    |   movel([0.097941, -1.446408, -2.526251, -0.739730, 1.570796, 1.668738],accel_mss,speed_ms,0,blend_radius_m)
    |   movel([0.099075, -1.445086, -2.527311, -0.739992, 1.570796, 1.669872],accel_mss,speed_ms,0,blend_radius_m)
    |   movel([0.103315, -1.440776, -2.530747, -0.740866, 1.570796, 1.674111],accel_mss,speed_ms,0,blend_radius_m)
    |   movel([0.107663, -1.436494, -2.534133, -0.741762, 1.570796, 1.678459],accel_mss,speed_ms,0,blend_radius_m)
    |   movel([0.104362, -1.438461, -2.532581, -0.741347, 1.570796, 1.675158],accel_mss,speed_ms,0,blend_radius_m)
    |   movel([0.101406, -1.440513, -2.530956, -0.740920, 1.570796, 1.672202],accel_mss,speed_ms,0,blend_radius_m)
    |   movel([0.098613, -1.442794, -2.529142, -0.740453, 1.570796, 1.669409],accel_mss,speed_ms,0,blend_radius_m)
    |   movel([0.095804, -1.445440, -2.527027, -0.739922, 1.570796, 1.666601],accel_mss,speed_ms,0,blend_radius_m)
    |   movel([0.097126, -1.443984, -2.528192, -0.740213, 1.570796, 1.667922],accel_mss,speed_ms,0,blend_radius_m)
    |   movel([0.098287, -1.442464, -2.529404, -0.740520, 1.570796, 1.669083],accel_mss,speed_ms,0,blend_radius_m)
    |   movel([0.102381, -1.436114, -2.534433, -0.741843, 1.570796, 1.673177],accel_mss,speed_ms,0,blend_radius_m)
    |   movel([0.103529, -1.434547, -2.535663, -0.742178, 1.570796, 1.674326],accel_mss,speed_ms,0,blend_radius_m)
    |   movel([0.104838, -1.433026, -2.536855, -0.742508, 1.570796, 1.675635],accel_mss,speed_ms,0,blend_radius_m)
    |   movel([0.106771, -1.431152, -2.538318, -0.742919, 1.570796, 1.677568],accel_mss,speed_ms,0,blend_radius_m)
    |   movel([0.108499, -1.429865, -2.539320, -0.743204, 1.570796, 1.679295],accel_mss,speed_ms,0,blend_radius_m)
    |   movel([0.108872, -1.429473, -2.539624, -0.743291, 1.570796, 1.679668],accel_mss,speed_ms,0,blend_radius_m)
    |   movel([0.108963, -1.429084, -2.539927, -0.743378, 1.570796, 1.679759],accel_mss,speed_ms,0,blend_radius_m)
    |   movel([0.108687, -1.428925, -2.540050, -0.743414, 1.570796, 1.679484],accel_mss,speed_ms,0,blend_radius_m)
    |   movel([0.108143, -1.428947, -2.540033, -0.743409, 1.570796, 1.678940],accel_mss,speed_ms,0,blend_radius_m)
    |   movel([0.107429, -1.429105, -2.539910, -0.743374, 1.570796, 1.678225],accel_mss,speed_ms,0,blend_radius_m)
    |   movel([0.105873, -1.429619, -2.539511, -0.743259, 1.570796, 1.676669],accel_mss,speed_ms,0,blend_radius_m)
    |   movel([0.104794, -1.430074, -2.539157, -0.743158, 1.570796, 1.675591],accel_mss,speed_ms,0,blend_radius_m)
    |   movel([0.106351, -1.428336, -2.540507, -0.743546, 1.570796, 1.677147],accel_mss,speed_ms,0,blend_radius_m)
    |   movel([0.108214, -1.426670, -2.541796, -0.743923, 1.570796, 1.679010],accel_mss,speed_ms,0,blend_radius_m)
    |   movel([0.112152, -1.423648, -2.544124, -0.744617, 1.570796, 1.682948],accel_mss,speed_ms,0,blend_radius_m)
    |   speed_ms = 0.005
    |   movel([0.112152, -1.415184, -2.540319, -0.756886, 1.570796, 1.682948],accel_mss,speed_ms,0,blend_radius_m)
    |   speed_ms = 0.040
    |   movel([0.104332, -1.417020, -2.538925, -0.756444, 1.570796, 1.675128],accel_mss,speed_ms,0,blend_radius_m)
    |   speed_ms = 0.005
    |   movel([0.104332, -1.425469, -2.542723, -0.744197, 1.570796, 1.675128],accel_mss,speed_ms,0,blend_radius_m)
    |   speed_ms = 0.025
    |   movel([0.103555, -1.424729, -2.543293, -0.744367, 1.570796, 1.674352],accel_mss,speed_ms,0,blend_radius_m)
    |   movel([0.102591, -1.424211, -2.543692, -0.744487, 1.570796, 1.673387],accel_mss,speed_ms,0,blend_radius_m)
    |   movel([0.101472, -1.423893, -2.543936, -0.744560, 1.570796, 1.672268],accel_mss,speed_ms,0,blend_radius_m)
    |   movel([0.100232, -1.423752, -2.544044, -0.744593, 1.570796, 1.671028],accel_mss,speed_ms,0,blend_radius_m)
    |   movel([0.098900, -1.423771, -2.544029, -0.744588, 1.570796, 1.669696],accel_mss,speed_ms,0,blend_radius_m)
    |   movel([0.097513, -1.423927, -2.543910, -0.744552, 1.570796, 1.668309],accel_mss,speed_ms,0,blend_radius_m)
    |   movel([0.094694, -1.424556, -2.543426, -0.744407, 1.570796, 1.665490],accel_mss,speed_ms,0,blend_radius_m)
    |   speed_ms = 0.005
    |   movel([0.094694, -1.416100, -2.539624, -0.756665, 1.570796, 1.665490],accel_mss,speed_ms,0,blend_radius_m)
    |   speed_ms = 0.040
    |   movel([0.105862, -1.410628, -2.543757, -0.758004, 1.570796, 1.676658],accel_mss,speed_ms,0,blend_radius_m)
    |   speed_ms = 0.005
    |   movel([0.105862, -1.419125, -2.547582, -0.745682, 1.570796, 1.676658],accel_mss,speed_ms,0,blend_radius_m)
    |   speed_ms = 0.025
    |   movel([0.105216, -1.417553, -2.548777, -0.746059, 1.570796, 1.676012],accel_mss,speed_ms,0,blend_radius_m)
    |   movel([0.104462, -1.416106, -2.549874, -0.746409, 1.570796, 1.675259],accel_mss,speed_ms,0,blend_radius_m)
    |   movel([0.103559, -1.414829, -2.550839, -0.746721, 1.570796, 1.674355],accel_mss,speed_ms,0,blend_radius_m)
    |   movel([0.102461, -1.413767, -2.551639, -0.746983, 1.570796, 1.673258],accel_mss,speed_ms,0,blend_radius_m)
    |   movel([0.101125, -1.412972, -2.552238, -0.747179, 1.570796, 1.671921],accel_mss,speed_ms,0,blend_radius_m)
    |   movel([0.099510, -1.412483, -2.552605, -0.747301, 1.570796, 1.670307],accel_mss,speed_ms,0,blend_radius_m)
    |   movel([0.097573, -1.412353, -2.552703, -0.747333, 1.570796, 1.668369],accel_mss,speed_ms,0,blend_radius_m)
    |   movel([0.096471, -1.412435, -2.552641, -0.747312, 1.570796, 1.667267],accel_mss,speed_ms,0,blend_radius_m)
    |   movel([0.095272, -1.412625, -2.552499, -0.747265, 1.570796, 1.666069],accel_mss,speed_ms,0,blend_radius_m)
    |   speed_ms = 0.005
    |   movel([0.095272, -1.404079, -2.548646, -0.759665, 1.570796, 1.666069],accel_mss,speed_ms,0,blend_radius_m)
    |   speed_ms = 0.040
    |   movel([0.104586, -1.399868, -2.551755, -0.760765, 1.570796, 1.675383],accel_mss,speed_ms,0,blend_radius_m)
    |   speed_ms = 0.005
    |   movel([0.104586, -1.408446, -2.555626, -0.748317, 1.570796, 1.675383],accel_mss,speed_ms,0,blend_radius_m)
    |   speed_ms = 0.025
    |   movel([0.103932, -1.404939, -2.558231, -0.749219, 1.570796, 1.674729],accel_mss,speed_ms,0,blend_radius_m)
    |   movel([0.103406, -1.403330, -2.559420, -0.749639, 1.570796, 1.674203],accel_mss,speed_ms,0,blend_radius_m)
    |   movel([0.102682, -1.401872, -2.560493, -0.750023, 1.570796, 1.673478],accel_mss,speed_ms,0,blend_radius_m)
    |   movel([0.101713, -1.400611, -2.561420, -0.750358, 1.570796, 1.672509],accel_mss,speed_ms,0,blend_radius_m)
    |   movel([0.100451, -1.399592, -2.562167, -0.750630, 1.570796, 1.671247],accel_mss,speed_ms,0,blend_radius_m)
    |   movel([0.098845, -1.398855, -2.562706, -0.750828, 1.570796, 1.669641],accel_mss,speed_ms,0,blend_radius_m)
    |   movel([0.096850, -1.398448, -2.563004, -0.750937, 1.570796, 1.667646],accel_mss,speed_ms,0,blend_radius_m)
    |   speed_ms = 0.005
    |   movel([0.096850, -1.389796, -2.559089, -0.763503, 1.570796, 1.667646],accel_mss,speed_ms,0,blend_radius_m)
    |   speed_ms = 0.040
    |   movel([0.105371, -1.389195, -2.559522, -0.763672, 1.570796, 1.676167],accel_mss,speed_ms,0,blend_radius_m)
    |   speed_ms = 0.005
    |   movel([0.105371, -1.397851, -2.563439, -0.751099, 1.570796, 1.676167],accel_mss,speed_ms,0,blend_radius_m)
    |   speed_ms = 0.025
    |   movel([0.105557, -1.395575, -2.565096, -0.751718, 1.570796, 1.676353],accel_mss,speed_ms,0,blend_radius_m)
    |   movel([0.105576, -1.393300, -2.566744, -0.752344, 1.570796, 1.676373],accel_mss,speed_ms,0,blend_radius_m)
    |   movel([0.105373, -1.391091, -2.568338, -0.752960, 1.570796, 1.676170],accel_mss,speed_ms,0,blend_radius_m)
    |   movel([0.104899, -1.389018, -2.569827, -0.753544, 1.570796, 1.675696],accel_mss,speed_ms,0,blend_radius_m)
    |   movel([0.104101, -1.387148, -2.571165, -0.754076, 1.570796, 1.674898],accel_mss,speed_ms,0,blend_radius_m)
    |   movel([0.103563, -1.386313, -2.571760, -0.754316, 1.570796, 1.674359],accel_mss,speed_ms,0,blend_radius_m)
    |   movel([0.102184, -1.384881, -2.572779, -0.754728, 1.570796, 1.672980],accel_mss,speed_ms,0,blend_radius_m)
    |   movel([0.101329, -1.384304, -2.573189, -0.754895, 1.570796, 1.672125],accel_mss,speed_ms,0,blend_radius_m)
    |   movel([0.100353, -1.383830, -2.573526, -0.755033, 1.570796, 1.671149],accel_mss,speed_ms,0,blend_radius_m)
    |   movel([0.099254, -1.383470, -2.573781, -0.755138, 1.570796, 1.670050],accel_mss,speed_ms,0,blend_radius_m)
    |   speed_ms = 0.005
    |   movel([0.099254, -1.374710, -2.569801, -0.767878, 1.570796, 1.670050],accel_mss,speed_ms,0,blend_radius_m)
    |   speed_ms = 0.040
    |   movel([0.108206, -1.373754, -2.570469, -0.768166, 1.570796, 1.679002],accel_mss,speed_ms,0,blend_radius_m)
    |   speed_ms = 0.005
    |   movel([0.108206, -1.382521, -2.574453, -0.755415, 1.570796, 1.679002],accel_mss,speed_ms,0,blend_radius_m)
    |   speed_ms = 0.025
    |   movel([0.108592, -1.379829, -2.576352, -0.756208, 1.570796, 1.679388],accel_mss,speed_ms,0,blend_radius_m)
    |   movel([0.108698, -1.377172, -2.578216, -0.757002, 1.570796, 1.679494],accel_mss,speed_ms,0,blend_radius_m)
    |   movel([0.108481, -1.374625, -2.579992, -0.757771, 1.570796, 1.679278],accel_mss,speed_ms,0,blend_radius_m)
    |   movel([0.107888, -1.372275, -2.581624, -0.758490, 1.570796, 1.678684],accel_mss,speed_ms,0,blend_radius_m)
    |   movel([0.106876, -1.370198, -2.583059, -0.759132, 1.570796, 1.677672],accel_mss,speed_ms,0,blend_radius_m)
    |   movel([0.106194, -1.369291, -2.583685, -0.759414, 1.570796, 1.676991],accel_mss,speed_ms,0,blend_radius_m)
    |   movel([0.105393, -1.368480, -2.584242, -0.759667, 1.570796, 1.676190],accel_mss,speed_ms,0,blend_radius_m)
    |   movel([0.104461, -1.367784, -2.584720, -0.759885, 1.570796, 1.675257],accel_mss,speed_ms,0,blend_radius_m)
    |   movel([0.103394, -1.367206, -2.585117, -0.760067, 1.570796, 1.674190],accel_mss,speed_ms,0,blend_radius_m)
    |   movel([0.102189, -1.366762, -2.585421, -0.760207, 1.570796, 1.672985],accel_mss,speed_ms,0,blend_radius_m)
    |   movel([0.100837, -1.366457, -2.585629, -0.760303, 1.570796, 1.671633],accel_mss,speed_ms,0,blend_radius_m)
    |   speed_ms = 0.005
    |   movel([0.100837, -1.357576, -2.581574, -0.773238, 1.570796, 1.671633],accel_mss,speed_ms,0,blend_radius_m)
    |   speed_ms = 0.040
    |   movel([0.059658, -1.369522, -2.573409, -0.769457, 1.570796, 1.630455],accel_mss,speed_ms,0,blend_radius_m)
    |   speed_ms = 0.005
    |   movel([0.059658, -1.378320, -2.577412, -0.756658, 1.570796, 1.630455],accel_mss,speed_ms,0,blend_radius_m)
    |   speed_ms = 0.025
    |   movel([0.061825, -1.379065, -2.576888, -0.756435, 1.570796, 1.632622],accel_mss,speed_ms,0,blend_radius_m)
    |   movel([0.063796, -1.380058, -2.576191, -0.756141, 1.570796, 1.634592],accel_mss,speed_ms,0,blend_radius_m)
    |   movel([0.065578, -1.381276, -2.575332, -0.755781, 1.570796, 1.636374],accel_mss,speed_ms,0,blend_radius_m)
    |   movel([0.067175, -1.382697, -2.574328, -0.755364, 1.570796, 1.637972],accel_mss,speed_ms,0,blend_radius_m)
    |   movel([0.068588, -1.384302, -2.573191, -0.754896, 1.570796, 1.639384],accel_mss,speed_ms,0,blend_radius_m)
    |   movel([0.069827, -1.386068, -2.571935, -0.754386, 1.570796, 1.640623],accel_mss,speed_ms,0,blend_radius_m)
    |   movel([0.070890, -1.387978, -2.570572, -0.753840, 1.570796, 1.641686],accel_mss,speed_ms,0,blend_radius_m)
    |   movel([0.071789, -1.390004, -2.569119, -0.753265, 1.570796, 1.642586],accel_mss,speed_ms,0,blend_radius_m)
    |   movel([0.072523, -1.392131, -2.567588, -0.752669, 1.570796, 1.643319],accel_mss,speed_ms,0,blend_radius_m)
    |   movel([0.073102, -1.394337, -2.565994, -0.752058, 1.570796, 1.643899],accel_mss,speed_ms,0,blend_radius_m)
    |   movel([0.073529, -1.396601, -2.564350, -0.751438, 1.570796, 1.644325],accel_mss,speed_ms,0,blend_radius_m)
    |   movel([0.073810, -1.398906, -2.562669, -0.750814, 1.570796, 1.644606],accel_mss,speed_ms,0,blend_radius_m)
    |   movel([0.073950, -1.401226, -2.560968, -0.750194, 1.570796, 1.644747],accel_mss,speed_ms,0,blend_radius_m)
    |   movel([0.073953, -1.403551, -2.559256, -0.749581, 1.570796, 1.644750],accel_mss,speed_ms,0,blend_radius_m)
    |   movel([0.073826, -1.405853, -2.557553, -0.748982, 1.570796, 1.644623],accel_mss,speed_ms,0,blend_radius_m)
    |   movel([0.073577, -1.408119, -2.555870, -0.748400, 1.570796, 1.644373],accel_mss,speed_ms,0,blend_radius_m)
    |   movel([0.073080, -1.411150, -2.553605, -0.747633, 1.570796, 1.643876],accel_mss,speed_ms,0,blend_radius_m)
    |   movel([0.072295, -1.414646, -2.550977, -0.746766, 1.570796, 1.643091],accel_mss,speed_ms,0,blend_radius_m)
    |   movel([0.071148, -1.418318, -2.548196, -0.745875, 1.570796, 1.641944],accel_mss,speed_ms,0,blend_radius_m)
    |   movel([0.070416, -1.420132, -2.546815, -0.745442, 1.570796, 1.641213],accel_mss,speed_ms,0,blend_radius_m)
    |   movel([0.069571, -1.421882, -2.545478, -0.745029, 1.570796, 1.640367],accel_mss,speed_ms,0,blend_radius_m)
    |   movel([0.068596, -1.423539, -2.544208, -0.744642, 1.570796, 1.639392],accel_mss,speed_ms,0,blend_radius_m)
    |   movel([0.067488, -1.425061, -2.543037, -0.744291, 1.570796, 1.638285],accel_mss,speed_ms,0,blend_radius_m)
    |   movel([0.066233, -1.426421, -2.541989, -0.743980, 1.570796, 1.637030],accel_mss,speed_ms,0,blend_radius_m)
    |   movel([0.064822, -1.427585, -2.541088, -0.743715, 1.570796, 1.635619],accel_mss,speed_ms,0,blend_radius_m)
    |   movel([0.063248, -1.428516, -2.540367, -0.743506, 1.570796, 1.634044],accel_mss,speed_ms,0,blend_radius_m)
    |   movel([0.061498, -1.429186, -2.539848, -0.743356, 1.570796, 1.632294],accel_mss,speed_ms,0,blend_radius_m)
    |   movel([0.060551, -1.429411, -2.539673, -0.743305, 1.570796, 1.631348],accel_mss,speed_ms,0,blend_radius_m)
    |   movel([0.059557, -1.429559, -2.539557, -0.743272, 1.570796, 1.630353],accel_mss,speed_ms,0,blend_radius_m)
    |   movel([0.057417, -1.429605, -2.539522, -0.743262, 1.570796, 1.628214],accel_mss,speed_ms,0,blend_radius_m)
    |   movel([0.054942, -1.429347, -2.539722, -0.743319, 1.570796, 1.625738],accel_mss,speed_ms,0,blend_radius_m)
    |   movel([0.052661, -1.428880, -2.540085, -0.743424, 1.570796, 1.623457],accel_mss,speed_ms,0,blend_radius_m)
    |   movel([0.050550, -1.428228, -2.540591, -0.743570, 1.570796, 1.621346],accel_mss,speed_ms,0,blend_radius_m)
    |   movel([0.048577, -1.427406, -2.541227, -0.743756, 1.570796, 1.619374],accel_mss,speed_ms,0,blend_radius_m)
    |   movel([0.046721, -1.426434, -2.541979, -0.743977, 1.570796, 1.617517],accel_mss,speed_ms,0,blend_radius_m)
    |   movel([0.044950, -1.425333, -2.542828, -0.744228, 1.570796, 1.615746],accel_mss,speed_ms,0,blend_radius_m)
    |   movel([0.041554, -1.422818, -2.544761, -0.744810, 1.570796, 1.612350],accel_mss,speed_ms,0,blend_radius_m)
    |   movel([0.037931, -1.419913, -2.546982, -0.745494, 1.570796, 1.608727],accel_mss,speed_ms,0,blend_radius_m)
    |   movel([0.034420, -1.416937, -2.549244, -0.746208, 1.570796, 1.605216],accel_mss,speed_ms,0,blend_radius_m)
    |   movel([0.031123, -1.413759, -2.551646, -0.746985, 1.570796, 1.601919],accel_mss,speed_ms,0,blend_radius_m)
    |   movel([0.029590, -1.412049, -2.552932, -0.747409, 1.570796, 1.600387],accel_mss,speed_ms,0,blend_radius_m)
    |   movel([0.028153, -1.410234, -2.554292, -0.747864, 1.570796, 1.598949],accel_mss,speed_ms,0,blend_radius_m)
    |   movel([0.026315, -1.408006, -2.555954, -0.748429, 1.570796, 1.597111],accel_mss,speed_ms,0,blend_radius_m)
    |   movel([0.024229, -1.405908, -2.557513, -0.748968, 1.570796, 1.595025],accel_mss,speed_ms,0,blend_radius_m)
    |   movel([0.021933, -1.403935, -2.558973, -0.749481, 1.570796, 1.592729],accel_mss,speed_ms,0,blend_radius_m)
    |   movel([0.019472, -1.402077, -2.560343, -0.749969, 1.570796, 1.590268],accel_mss,speed_ms,0,blend_radius_m)
    |   movel([0.014218, -1.398680, -2.562834, -0.750875, 1.570796, 1.585014],accel_mss,speed_ms,0,blend_radius_m)
    |   movel([0.008809, -1.395643, -2.565047, -0.751699, 1.570796, 1.579605],accel_mss,speed_ms,0,blend_radius_m)
    |   movel([0.004540, -1.393597, -2.566530, -0.752262, 1.570796, 1.575336],accel_mss,speed_ms,0,blend_radius_m)
    |   movel([-0.000022, -1.391895, -2.567759, -0.752735, 1.570796, 1.570774],accel_mss,speed_ms,0,blend_radius_m)
    |   movel([-0.004863, -1.390560, -2.568720, -0.753109, 1.570796, 1.565933],accel_mss,speed_ms,0,blend_radius_m)
    |   movel([-0.009964, -1.389616, -2.569398, -0.753375, 1.570796, 1.560832],accel_mss,speed_ms,0,blend_radius_m)
    |   movel([-0.015307, -1.389081, -2.569782, -0.753526, 1.570796, 1.555489],accel_mss,speed_ms,0,blend_radius_m)
    |   movel([-0.018062, -1.388974, -2.569859, -0.753557, 1.570796, 1.552735],accel_mss,speed_ms,0,blend_radius_m)
    |   movel([-0.023729, -1.389089, -2.569776, -0.753524, 1.570796, 1.547068],accel_mss,speed_ms,0,blend_radius_m)
    |   movel([-0.026636, -1.389317, -2.569612, -0.753459, 1.570796, 1.544160],accel_mss,speed_ms,0,blend_radius_m)
    |   movel([-0.032578, -1.390124, -2.569034, -0.753232, 1.570796, 1.538218],accel_mss,speed_ms,0,blend_radius_m)
    |   movel([-0.036711, -1.390995, -2.568408, -0.752987, 1.570796, 1.534085],accel_mss,speed_ms,0,blend_radius_m)
    |   movel([-0.040890, -1.392189, -2.567547, -0.752653, 1.570796, 1.529906],accel_mss,speed_ms,0,blend_radius_m)
    |   movel([-0.045076, -1.393696, -2.566458, -0.752235, 1.570796, 1.525721],accel_mss,speed_ms,0,blend_radius_m)
    |   movel([-0.049230, -1.395512, -2.565142, -0.751735, 1.570796, 1.521566],accel_mss,speed_ms,0,blend_radius_m)
    |   movel([-0.053319, -1.397627, -2.563602, -0.751159, 1.570796, 1.517478],accel_mss,speed_ms,0,blend_radius_m)
    |   movel([-0.057302, -1.400033, -2.561844, -0.750512, 1.570796, 1.513494],accel_mss,speed_ms,0,blend_radius_m)
    |   movel([-0.061143, -1.402719, -2.559870, -0.749800, 1.570796, 1.509653],accel_mss,speed_ms,0,blend_radius_m)
    |   movel([-0.064808, -1.405675, -2.557686, -0.749028, 1.570796, 1.505989],accel_mss,speed_ms,0,blend_radius_m)
    |   movel([-0.068038, -1.408621, -2.555496, -0.748272, 1.570796, 1.502758],accel_mss,speed_ms,0,blend_radius_m)
    |   movel([-0.070971, -1.411618, -2.553255, -0.747516, 1.570796, 1.499825],accel_mss,speed_ms,0,blend_radius_m)
    |   movel([-0.073584, -1.414666, -2.550962, -0.746761, 1.570796, 1.497212],accel_mss,speed_ms,0,blend_radius_m)
    |   movel([-0.075859, -1.417769, -2.548613, -0.746007, 1.570796, 1.494937],accel_mss,speed_ms,0,blend_radius_m)
    |   movel([-0.076864, -1.419343, -2.547417, -0.745630, 1.570796, 1.493932],accel_mss,speed_ms,0,blend_radius_m)
    |   movel([-0.078594, -1.422530, -2.544981, -0.744877, 1.570796, 1.492203],accel_mss,speed_ms,0,blend_radius_m)
    |   movel([-0.079313, -1.424148, -2.543740, -0.744501, 1.570796, 1.491483],accel_mss,speed_ms,0,blend_radius_m)
    |   movel([-0.080451, -1.427426, -2.541212, -0.743751, 1.570796, 1.490346],accel_mss,speed_ms,0,blend_radius_m)
    |   movel([-0.080865, -1.429090, -2.539922, -0.743377, 1.570796, 1.489931],accel_mss,speed_ms,0,blend_radius_m)
    |   movel([-0.081172, -1.430768, -2.538618, -0.743004, 1.570796, 1.489624],accel_mss,speed_ms,0,blend_radius_m)
    |   movel([-0.081449, -1.433150, -2.536758, -0.742481, 1.570796, 1.489347],accel_mss,speed_ms,0,blend_radius_m)
    |   movel([-0.081564, -1.435509, -2.534908, -0.741972, 1.570796, 1.489232],accel_mss,speed_ms,0,blend_radius_m)
    |   movel([-0.081528, -1.437829, -2.533080, -0.741479, 1.570796, 1.489268],accel_mss,speed_ms,0,blend_radius_m)
    |   movel([-0.081354, -1.440107, -2.531278, -0.741004, 1.570796, 1.489442],accel_mss,speed_ms,0,blend_radius_m)
    |   movel([-0.081048, -1.442324, -2.529516, -0.740549, 1.570796, 1.489748],accel_mss,speed_ms,0,blend_radius_m)
    |   movel([-0.080619, -1.444471, -2.527803, -0.740115, 1.570796, 1.490177],accel_mss,speed_ms,0,blend_radius_m)
    |   movel([-0.080080, -1.446539, -2.526146, -0.739704, 1.570796, 1.490717],accel_mss,speed_ms,0,blend_radius_m)
    |   movel([-0.079436, -1.448513, -2.524558, -0.739318, 1.570796, 1.491360],accel_mss,speed_ms,0,blend_radius_m)
    |   movel([-0.076104, -1.455825, -2.518624, -0.737940, 1.570796, 1.494693],accel_mss,speed_ms,0,blend_radius_m)
    |   movel([-0.073504, -1.461704, -2.513794, -0.736892, 1.570796, 1.497293],accel_mss,speed_ms,0,blend_radius_m)
    |   movel([-0.073326, -1.462294, -2.513305, -0.736790, 1.570796, 1.497470],accel_mss,speed_ms,0,blend_radius_m)
    |   movel([-0.069320, -1.459022, -2.516004, -0.737363, 1.570796, 1.501476],accel_mss,speed_ms,0,blend_radius_m)
    |   movel([-0.065110, -1.455930, -2.518539, -0.737921, 1.570796, 1.505686],accel_mss,speed_ms,0,blend_radius_m)
    |   movel([-0.060722, -1.453023, -2.520907, -0.738458, 1.570796, 1.510074],accel_mss,speed_ms,0,blend_radius_m)
    |   movel([-0.056193, -1.450309, -2.523108, -0.738972, 1.570796, 1.514604],accel_mss,speed_ms,0,blend_radius_m)
    |   movel([-0.051554, -1.447796, -2.525135, -0.739458, 1.570796, 1.519242],accel_mss,speed_ms,0,blend_radius_m)
    |   movel([-0.046842, -1.445487, -2.526990, -0.739913, 1.570796, 1.523955],accel_mss,speed_ms,0,blend_radius_m)
    |   movel([-0.042089, -1.443391, -2.528665, -0.740332, 1.570796, 1.528708],accel_mss,speed_ms,0,blend_radius_m)
    |   movel([-0.037332, -1.441513, -2.530162, -0.740715, 1.570796, 1.533464],accel_mss,speed_ms,0,blend_radius_m)
    |   movel([-0.035087, -1.440732, -2.530782, -0.740875, 1.570796, 1.535710],accel_mss,speed_ms,0,blend_radius_m)
    |   movel([-0.032797, -1.440048, -2.531325, -0.741016, 1.570796, 1.537999],accel_mss,speed_ms,0,blend_radius_m)
    |   movel([-0.030483, -1.439471, -2.531782, -0.741136, 1.570796, 1.540314],accel_mss,speed_ms,0,blend_radius_m)
    |   movel([-0.028168, -1.439011, -2.532146, -0.741232, 1.570796, 1.542628],accel_mss,speed_ms,0,blend_radius_m)
    |   movel([-0.025873, -1.438678, -2.532410, -0.741301, 1.570796, 1.544923],accel_mss,speed_ms,0,blend_radius_m)
    |   movel([-0.023617, -1.438482, -2.532564, -0.741342, 1.570796, 1.547179],accel_mss,speed_ms,0,blend_radius_m)
    |   movel([-0.021423, -1.438432, -2.532604, -0.741353, 1.570796, 1.549374],accel_mss,speed_ms,0,blend_radius_m)
    |   movel([-0.019312, -1.438537, -2.532521, -0.741331, 1.570796, 1.551485],accel_mss,speed_ms,0,blend_radius_m)
    |   movel([-0.017304, -1.438806, -2.532308, -0.741275, 1.570796, 1.553492],accel_mss,speed_ms,0,blend_radius_m)
    |   movel([-0.015419, -1.439248, -2.531958, -0.741182, 1.570796, 1.555377],accel_mss,speed_ms,0,blend_radius_m)
    |   movel([-0.013682, -1.439873, -2.531463, -0.741052, 1.570796, 1.557115],accel_mss,speed_ms,0,blend_radius_m)
    |   movel([-0.012110, -1.440688, -2.530817, -0.740884, 1.570796, 1.558686],accel_mss,speed_ms,0,blend_radius_m)
    |   movel([-0.010727, -1.441700, -2.530013, -0.740676, 1.570796, 1.560070],accel_mss,speed_ms,0,blend_radius_m)
    |   movel([-0.009547, -1.442918, -2.529043, -0.740428, 1.570796, 1.561249],accel_mss,speed_ms,0,blend_radius_m)
    |   movel([-0.008594, -1.444348, -2.527901, -0.740140, 1.570796, 1.562202],accel_mss,speed_ms,0,blend_radius_m)
    |   movel([-0.007889, -1.445999, -2.526579, -0.739811, 1.570796, 1.562907],accel_mss,speed_ms,0,blend_radius_m)
    |   movel([-0.007322, -1.448381, -2.524664, -0.739344, 1.570796, 1.563474],accel_mss,speed_ms,0,blend_radius_m)
    |   movel([-0.007078, -1.450952, -2.522588, -0.738849, 1.570796, 1.563718],accel_mss,speed_ms,0,blend_radius_m)
    |   movel([-0.007113, -1.453662, -2.520388, -0.738339, 1.570796, 1.563684],accel_mss,speed_ms,0,blend_radius_m)
    |   movel([-0.007377, -1.456466, -2.518100, -0.737823, 1.570796, 1.563419],accel_mss,speed_ms,0,blend_radius_m)
    |   movel([-0.007828, -1.459313, -2.515764, -0.737312, 1.570796, 1.562969],accel_mss,speed_ms,0,blend_radius_m)
    |   movel([-0.008422, -1.462161, -2.513416, -0.736813, 1.570796, 1.562374],accel_mss,speed_ms,0,blend_radius_m)
    |   movel([-0.009854, -1.467669, -2.508837, -0.735883, 1.570796, 1.560943],accel_mss,speed_ms,0,blend_radius_m)
    |   movel([-0.010947, -1.471129, -2.505936, -0.735324, 1.570796, 1.559849],accel_mss,speed_ms,0,blend_radius_m)
    |   movel([-0.012225, -1.474530, -2.503067, -0.734792, 1.570796, 1.558571],accel_mss,speed_ms,0,blend_radius_m)
    |   movel([-0.013665, -1.477882, -2.500222, -0.734285, 1.570796, 1.557131],accel_mss,speed_ms,0,blend_radius_m)
    |   movel([-0.015247, -1.481200, -2.497388, -0.733801, 1.570796, 1.555549],accel_mss,speed_ms,0,blend_radius_m)
    |   movel([-0.016950, -1.484491, -2.494559, -0.733338, 1.570796, 1.553847],accel_mss,speed_ms,0,blend_radius_m)
    |   movel([-0.018751, -1.487769, -2.491725, -0.732894, 1.570796, 1.552045],accel_mss,speed_ms,0,blend_radius_m)
    |   movel([-0.022580, -1.494335, -2.485998, -0.732056, 1.570796, 1.548217],accel_mss,speed_ms,0,blend_radius_m)
    |   movel([-0.019141, -1.495499, -2.484976, -0.731914, 1.570796, 1.551655],accel_mss,speed_ms,0,blend_radius_m)
    |   movel([-0.017373, -1.496216, -2.484345, -0.731828, 1.570796, 1.553424],accel_mss,speed_ms,0,blend_radius_m)
    |   movel([-0.015874, -1.497092, -2.483573, -0.731724, 1.570796, 1.554922],accel_mss,speed_ms,0,blend_radius_m)
    |   movel([-0.015298, -1.497607, -2.483119, -0.731663, 1.570796, 1.555498],accel_mss,speed_ms,0,blend_radius_m)
    |   movel([-0.014876, -1.498181, -2.482612, -0.731596, 1.570796, 1.555921],accel_mss,speed_ms,0,blend_radius_m)
    |   movel([-0.014633, -1.498821, -2.482046, -0.731522, 1.570796, 1.556163],accel_mss,speed_ms,0,blend_radius_m)
    |   movel([-0.014598, -1.499532, -2.481417, -0.731440, 1.570796, 1.556198],accel_mss,speed_ms,0,blend_radius_m)
    |   movel([-0.014799, -1.500318, -2.480720, -0.731351, 1.570796, 1.555997],accel_mss,speed_ms,0,blend_radius_m)
    |   movel([-0.015266, -1.501190, -2.479946, -0.731253, 1.570796, 1.555531],accel_mss,speed_ms,0,blend_radius_m)
    |   movel([-0.016023, -1.502154, -2.479089, -0.731146, 1.570796, 1.554774],accel_mss,speed_ms,0,blend_radius_m)
    |   movel([-0.017098, -1.503212, -2.478147, -0.731030, 1.570796, 1.553698],accel_mss,speed_ms,0,blend_radius_m)
    |   movel([-0.018095, -1.504041, -2.477407, -0.730941, 1.570796, 1.552701],accel_mss,speed_ms,0,blend_radius_m)
    |   movel([-0.019098, -1.504759, -2.476766, -0.730864, 1.570796, 1.551698],accel_mss,speed_ms,0,blend_radius_m)
    |   movel([-0.020104, -1.505374, -2.476216, -0.730799, 1.570796, 1.550693],accel_mss,speed_ms,0,blend_radius_m)
    |   movel([-0.022128, -1.506331, -2.475359, -0.730700, 1.570796, 1.548668],accel_mss,speed_ms,0,blend_radius_m)
    |   movel([-0.023145, -1.506690, -2.475037, -0.730663, 1.570796, 1.547651],accel_mss,speed_ms,0,blend_radius_m)
    |   movel([-0.025190, -1.507214, -2.474566, -0.730609, 1.570796, 1.545607],accel_mss,speed_ms,0,blend_radius_m)
    |   movel([-0.027240, -1.507536, -2.474277, -0.730576, 1.570796, 1.543556],accel_mss,speed_ms,0,blend_radius_m)
    |   movel([-0.029296, -1.507724, -2.474108, -0.730557, 1.570796, 1.541501],accel_mss,speed_ms,0,blend_radius_m)
    |   movel([-0.033399, -1.507966, -2.473890, -0.730533, 1.570796, 1.537397],accel_mss,speed_ms,0,blend_radius_m)
    |   movel([-0.035635, -1.510509, -2.471599, -0.730281, 1.570796, 1.535161],accel_mss,speed_ms,0,blend_radius_m)
    |   movel([-0.036859, -1.511755, -2.470472, -0.730162, 1.570796, 1.533937],accel_mss,speed_ms,0,blend_radius_m)
    |   movel([-0.038156, -1.512939, -2.469399, -0.730051, 1.570796, 1.532640],accel_mss,speed_ms,0,blend_radius_m)
    |   movel([-0.039530, -1.514027, -2.468412, -0.729950, 1.570796, 1.531267],accel_mss,speed_ms,0,blend_radius_m)
    |   movel([-0.040978, -1.514982, -2.467543, -0.729864, 1.570796, 1.529818],accel_mss,speed_ms,0,blend_radius_m)
    |   movel([-0.042505, -1.515772, -2.466824, -0.729794, 1.570796, 1.528291],accel_mss,speed_ms,0,blend_radius_m)
    |   movel([-0.044115, -1.516362, -2.466285, -0.729742, 1.570796, 1.526681],accel_mss,speed_ms,0,blend_radius_m)
    |   movel([-0.045238, -1.516569, -2.466096, -0.729724, 1.570796, 1.525558],accel_mss,speed_ms,0,blend_radius_m)
    |   movel([-0.046116, -1.516495, -2.466164, -0.729730, 1.570796, 1.524681],accel_mss,speed_ms,0,blend_radius_m)
    |   movel([-0.046775, -1.516183, -2.466449, -0.729757, 1.570796, 1.524022],accel_mss,speed_ms,0,blend_radius_m)
    |   movel([-0.047239, -1.515675, -2.466912, -0.729802, 1.570796, 1.523558],accel_mss,speed_ms,0,blend_radius_m)
    |   movel([-0.047533, -1.515013, -2.467515, -0.729861, 1.570796, 1.523263],accel_mss,speed_ms,0,blend_radius_m)
    |   movel([-0.047682, -1.514245, -2.468213, -0.729930, 1.570796, 1.523114],accel_mss,speed_ms,0,blend_radius_m)
    |   movel([-0.047712, -1.513411, -2.468971, -0.730007, 1.570796, 1.523084],accel_mss,speed_ms,0,blend_radius_m)
    |   movel([-0.047643, -1.512554, -2.469748, -0.730086, 1.570796, 1.523154],accel_mss,speed_ms,0,blend_radius_m)
    |   movel([-0.047294, -1.510714, -2.471413, -0.730261, 1.570796, 1.523503],accel_mss,speed_ms,0,blend_radius_m)
    |   movel([-0.046752, -1.508869, -2.473078, -0.730442, 1.570796, 1.524045],accel_mss,speed_ms,0,blend_radius_m)
    |   movel([-0.045381, -1.505113, -2.476449, -0.730827, 1.570796, 1.525416],accel_mss,speed_ms,0,blend_radius_m)
    |   movel([-0.049954, -1.502992, -2.478343, -0.731054, 1.570796, 1.520842],accel_mss,speed_ms,0,blend_radius_m)
    |   movel([-0.054648, -1.500999, -2.480116, -0.731274, 1.570796, 1.516149],accel_mss,speed_ms,0,blend_radius_m)
    |   movel([-0.059326, -1.498967, -2.481917, -0.731505, 1.570796, 1.511471],accel_mss,speed_ms,0,blend_radius_m)
    |   movel([-0.061617, -1.497884, -2.482875, -0.731631, 1.570796, 1.509179],accel_mss,speed_ms,0,blend_radius_m)
    |   movel([-0.063856, -1.496726, -2.483896, -0.731767, 1.570796, 1.506941],accel_mss,speed_ms,0,blend_radius_m)
    |   movel([-0.065924, -1.495528, -2.484950, -0.731910, 1.570796, 1.504873],accel_mss,speed_ms,0,blend_radius_m)
    |   movel([-0.067906, -1.494259, -2.486065, -0.732065, 1.570796, 1.502890],accel_mss,speed_ms,0,blend_radius_m)
    |   movel([-0.071708, -1.491577, -2.488412, -0.732400, 1.570796, 1.499088],accel_mss,speed_ms,0,blend_radius_m)
    |   movel([-0.075462, -1.488851, -2.490787, -0.732751, 1.570796, 1.495334],accel_mss,speed_ms,0,blend_radius_m)
    |   movel([-0.079361, -1.486249, -2.493042, -0.733098, 1.570796, 1.491435],accel_mss,speed_ms,0,blend_radius_m)
    |   movel([-0.080463, -1.488354, -2.491218, -0.732817, 1.570796, 1.490333],accel_mss,speed_ms,0,blend_radius_m)
    |   movel([-0.081432, -1.490449, -2.489396, -0.732544, 1.570796, 1.489365],accel_mss,speed_ms,0,blend_radius_m)
    |   movel([-0.082267, -1.492529, -2.487581, -0.732279, 1.570796, 1.488530],accel_mss,speed_ms,0,blend_radius_m)
    |   movel([-0.082969, -1.494588, -2.485777, -0.732025, 1.570796, 1.487827],accel_mss,speed_ms,0,blend_radius_m)
    |   movel([-0.083539, -1.496624, -2.483986, -0.731779, 1.570796, 1.487258],accel_mss,speed_ms,0,blend_radius_m)
    |   movel([-0.083978, -1.498631, -2.482215, -0.731544, 1.570796, 1.486818],accel_mss,speed_ms,0,blend_radius_m)
    |   movel([-0.084285, -1.500606, -2.480465, -0.731318, 1.570796, 1.486511],accel_mss,speed_ms,0,blend_radius_m)
    |   movel([-0.084466, -1.502546, -2.478740, -0.731103, 1.570796, 1.486331],accel_mss,speed_ms,0,blend_radius_m)
    |   movel([-0.084516, -1.504447, -2.477045, -0.730898, 1.570796, 1.486280],accel_mss,speed_ms,0,blend_radius_m)
    |   movel([-0.084436, -1.506303, -2.475383, -0.730703, 1.570796, 1.486361],accel_mss,speed_ms,0,blend_radius_m)
    |   movel([-0.084230, -1.508115, -2.473757, -0.730518, 1.570796, 1.486566],accel_mss,speed_ms,0,blend_radius_m)
    |   movel([-0.083899, -1.509875, -2.472171, -0.730343, 1.570796, 1.486898],accel_mss,speed_ms,0,blend_radius_m)
    |   movel([-0.083438, -1.511581, -2.470630, -0.730178, 1.570796, 1.487358],accel_mss,speed_ms,0,blend_radius_m)
    |   movel([-0.082854, -1.513231, -2.469135, -0.730023, 1.570796, 1.487942],accel_mss,speed_ms,0,blend_radius_m)
    |   movel([-0.082145, -1.514819, -2.467691, -0.729879, 1.570796, 1.488651],accel_mss,speed_ms,0,blend_radius_m)
    |   movel([-0.081311, -1.516345, -2.466301, -0.729743, 1.570796, 1.489485],accel_mss,speed_ms,0,blend_radius_m)
    |   movel([-0.079795, -1.518566, -2.464270, -0.729553, 1.570796, 1.491001],accel_mss,speed_ms,0,blend_radius_m)
    |   movel([-0.078055, -1.520599, -2.462405, -0.729385, 1.570796, 1.492742],accel_mss,speed_ms,0,blend_radius_m)
    |   movel([-0.076117, -1.522459, -2.460692, -0.729238, 1.570796, 1.494679],accel_mss,speed_ms,0,blend_radius_m)
    |   movel([-0.074001, -1.524162, -2.459119, -0.729108, 1.570796, 1.496795],accel_mss,speed_ms,0,blend_radius_m)
    |   movel([-0.071735, -1.525724, -2.457672, -0.728993, 1.570796, 1.499062],accel_mss,speed_ms,0,blend_radius_m)
    |   movel([-0.069341, -1.527159, -2.456340, -0.728890, 1.570796, 1.501456],accel_mss,speed_ms,0,blend_radius_m)
    |   movel([-0.066843, -1.528483, -2.455108, -0.728799, 1.570796, 1.503953],accel_mss,speed_ms,0,blend_radius_m)
    |   movel([-0.064261, -1.529706, -2.453967, -0.728716, 1.570796, 1.506535],accel_mss,speed_ms,0,blend_radius_m)
    |   movel([-0.058915, -1.531954, -2.451863, -0.728572, 1.570796, 1.511882],accel_mss,speed_ms,0,blend_radius_m)
    |   movel([-0.053475, -1.534068, -2.449878, -0.728443, 1.570796, 1.517321],accel_mss,speed_ms,0,blend_radius_m)
    |   movel([-0.049350, -1.535795, -2.448251, -0.728343, 1.570796, 1.521446],accel_mss,speed_ms,0,blend_radius_m)
    |   movel([-0.047922, -1.536279, -2.447794, -0.728316, 1.570796, 1.522874],accel_mss,speed_ms,0,blend_radius_m)
    |   movel([-0.045334, -1.536940, -2.447169, -0.728280, 1.570796, 1.525463],accel_mss,speed_ms,0,blend_radius_m)
    |   movel([-0.044798, -1.537178, -2.446944, -0.728267, 1.570796, 1.525998],accel_mss,speed_ms,0,blend_radius_m)
    |   movel([-0.044322, -1.537503, -2.446637, -0.728250, 1.570796, 1.526475],accel_mss,speed_ms,0,blend_radius_m)
    |   movel([-0.043916, -1.537944, -2.446219, -0.728226, 1.570796, 1.526880],accel_mss,speed_ms,0,blend_radius_m)
    |   movel([-0.043592, -1.538530, -2.445663, -0.728195, 1.570796, 1.527205],accel_mss,speed_ms,0,blend_radius_m)
    |   movel([-0.043368, -1.539293, -2.444940, -0.728156, 1.570796, 1.527428],accel_mss,speed_ms,0,blend_radius_m)
    |   movel([-0.043314, -1.540103, -2.444171, -0.728116, 1.570796, 1.527483],accel_mss,speed_ms,0,blend_radius_m)
    |   movel([-0.043411, -1.540949, -2.443366, -0.728074, 1.570796, 1.527385],accel_mss,speed_ms,0,blend_radius_m)
    |   movel([-0.043649, -1.541827, -2.442530, -0.728033, 1.570796, 1.527148],accel_mss,speed_ms,0,blend_radius_m)
    |   movel([-0.044011, -1.542723, -2.441675, -0.727991, 1.570796, 1.526786],accel_mss,speed_ms,0,blend_radius_m)
    |   movel([-0.045056, -1.544546, -2.439931, -0.727912, 1.570796, 1.525740],accel_mss,speed_ms,0,blend_radius_m)
    |   movel([-0.045713, -1.545455, -2.439061, -0.727874, 1.570796, 1.525083],accel_mss,speed_ms,0,blend_radius_m)
    |   movel([-0.047218, -1.547224, -2.437361, -0.727804, 1.570796, 1.523578],accel_mss,speed_ms,0,blend_radius_m)
    |   movel([-0.048899, -1.548876, -2.435770, -0.727744, 1.570796, 1.521898],accel_mss,speed_ms,0,blend_radius_m)
    |   movel([-0.050641, -1.550343, -2.434352, -0.727694, 1.570796, 1.520155],accel_mss,speed_ms,0,blend_radius_m)
    |   movel([-0.052345, -1.551562, -2.433172, -0.727655, 1.570796, 1.518451],accel_mss,speed_ms,0,blend_radius_m)
    |   movel([-0.055003, -1.553125, -2.431656, -0.727608, 1.570796, 1.515794],accel_mss,speed_ms,0,blend_radius_m)
    |   movel([-0.056377, -1.553814, -2.430986, -0.727589, 1.570796, 1.514419],accel_mss,speed_ms,0,blend_radius_m)
    |   movel([-0.057771, -1.554438, -2.430379, -0.727572, 1.570796, 1.513025],accel_mss,speed_ms,0,blend_radius_m)
    |   movel([-0.060603, -1.555491, -2.429353, -0.727545, 1.570796, 1.510193],accel_mss,speed_ms,0,blend_radius_m)
    |   movel([-0.063453, -1.556276, -2.428587, -0.727526, 1.570796, 1.507344],accel_mss,speed_ms,0,blend_radius_m)
    |   movel([-0.066275, -1.556782, -2.428092, -0.727515, 1.570796, 1.504521],accel_mss,speed_ms,0,blend_radius_m)
    |   movel([-0.069020, -1.557000, -2.427879, -0.727510, 1.570796, 1.501776],accel_mss,speed_ms,0,blend_radius_m)
    |   movel([-0.070351, -1.556996, -2.427883, -0.727510, 1.570796, 1.500445],accel_mss,speed_ms,0,blend_radius_m)
    |   movel([-0.072900, -1.556759, -2.428115, -0.727515, 1.570796, 1.497896],accel_mss,speed_ms,0,blend_radius_m)
    |   movel([-0.074106, -1.556521, -2.428347, -0.727521, 1.570796, 1.496690],accel_mss,speed_ms,0,blend_radius_m)
    |   movel([-0.075629, -1.556091, -2.428768, -0.727531, 1.570796, 1.495168],accel_mss,speed_ms,0,blend_radius_m)
    |   movel([-0.077066, -1.555548, -2.429297, -0.727544, 1.570796, 1.493731],accel_mss,speed_ms,0,blend_radius_m)
    |   movel([-0.078425, -1.554908, -2.429921, -0.727560, 1.570796, 1.492372],accel_mss,speed_ms,0,blend_radius_m)
    |   movel([-0.079719, -1.554187, -2.430624, -0.727579, 1.570796, 1.491077],accel_mss,speed_ms,0,blend_radius_m)
    |   movel([-0.082152, -1.552560, -2.432204, -0.727624, 1.570796, 1.488644],accel_mss,speed_ms,0,blend_radius_m)
    |   movel([-0.084447, -1.550793, -2.433917, -0.727679, 1.570796, 1.486349],accel_mss,speed_ms,0,blend_radius_m)
    |   movel([-0.087214, -1.548474, -2.436157, -0.727758, 1.570796, 1.483583],accel_mss,speed_ms,0,blend_radius_m)
    |   movel([-0.089858, -1.546009, -2.438528, -0.727852, 1.570796, 1.480939],accel_mss,speed_ms,0,blend_radius_m)
    |   movel([-0.092354, -1.543396, -2.441032, -0.727961, 1.570796, 1.478443],accel_mss,speed_ms,0,blend_radius_m)
    |   movel([-0.094679, -1.540631, -2.443668, -0.728090, 1.570796, 1.476118],accel_mss,speed_ms,0,blend_radius_m)
    |   movel([-0.096807, -1.537710, -2.446441, -0.728238, 1.570796, 1.473989],accel_mss,speed_ms,0,blend_radius_m)
    |   movel([-0.098711, -1.534629, -2.449349, -0.728410, 1.570796, 1.472086],accel_mss,speed_ms,0,blend_radius_m)
    |   movel([-0.100365, -1.531386, -2.452395, -0.728608, 1.570796, 1.470431],accel_mss,speed_ms,0,blend_radius_m)
    |   movel([-0.101745, -1.527976, -2.455580, -0.728833, 1.570796, 1.469052],accel_mss,speed_ms,0,blend_radius_m)
    |   movel([-0.102598, -1.525304, -2.458061, -0.729023, 1.570796, 1.468199],accel_mss,speed_ms,0,blend_radius_m)
    |   movel([-0.103327, -1.522453, -2.460698, -0.729238, 1.570796, 1.467470],accel_mss,speed_ms,0,blend_radius_m)
    |   movel([-0.103895, -1.519449, -2.463461, -0.729479, 1.570796, 1.466901],accel_mss,speed_ms,0,blend_radius_m)
    |   movel([-0.104269, -1.516327, -2.466317, -0.729745, 1.570796, 1.466527],accel_mss,speed_ms,0,blend_radius_m)
    |   movel([-0.104412, -1.513119, -2.469236, -0.730034, 1.570796, 1.466384],accel_mss,speed_ms,0,blend_radius_m)
    |   movel([-0.104286, -1.509858, -2.472187, -0.730345, 1.570796, 1.466511],accel_mss,speed_ms,0,blend_radius_m)
    |   movel([-0.103856, -1.506574, -2.475141, -0.730675, 1.570796, 1.466940],accel_mss,speed_ms,0,blend_radius_m)
    |   movel([-0.103514, -1.504934, -2.476609, -0.730846, 1.570796, 1.467282],accel_mss,speed_ms,0,blend_radius_m)
    |   movel([-0.103083, -1.503302, -2.478066, -0.731020, 1.570796, 1.467714],accel_mss,speed_ms,0,blend_radius_m)
    |   movel([-0.102065, -1.500231, -2.480797, -0.731361, 1.570796, 1.468731],accel_mss,speed_ms,0,blend_radius_m)
    |   movel([-0.100816, -1.497139, -2.483531, -0.731718, 1.570796, 1.469980],accel_mss,speed_ms,0,blend_radius_m)
    |   movel([-0.099340, -1.494040, -2.486258, -0.732092, 1.570796, 1.471456],accel_mss,speed_ms,0,blend_radius_m)
    |   movel([-0.097645, -1.490946, -2.488963, -0.732480, 1.570796, 1.473151],accel_mss,speed_ms,0,blend_radius_m)
    |   movel([-0.095732, -1.487871, -2.491638, -0.732881, 1.570796, 1.475065],accel_mss,speed_ms,0,blend_radius_m)
    |   movel([-0.093611, -1.484830, -2.494267, -0.733292, 1.570796, 1.477185],accel_mss,speed_ms,0,blend_radius_m)
    |   movel([-0.091286, -1.481838, -2.496841, -0.733710, 1.570796, 1.479510],accel_mss,speed_ms,0,blend_radius_m)
    |   movel([-0.088762, -1.478910, -2.499346, -0.734134, 1.570796, 1.482034],accel_mss,speed_ms,0,blend_radius_m)
    |   movel([-0.092940, -1.473333, -2.504079, -0.734977, 1.570796, 1.477856],accel_mss,speed_ms,0,blend_radius_m)
    |   movel([-0.095041, -1.470536, -2.506435, -0.735418, 1.570796, 1.475755],accel_mss,speed_ms,0,blend_radius_m)
    |   movel([-0.097004, -1.467625, -2.508873, -0.735890, 1.570796, 1.473792],accel_mss,speed_ms,0,blend_radius_m)
    |   movel([-0.098264, -1.465308, -2.510805, -0.736276, 1.570796, 1.472533],accel_mss,speed_ms,0,blend_radius_m)
    |   movel([-0.099276, -1.462829, -2.512862, -0.736697, 1.570796, 1.471520],accel_mss,speed_ms,0,blend_radius_m)
    |   movel([-0.100052, -1.460205, -2.515030, -0.737154, 1.570796, 1.470745],accel_mss,speed_ms,0,blend_radius_m)
    |   movel([-0.100596, -1.457445, -2.517298, -0.737646, 1.570796, 1.470200],accel_mss,speed_ms,0,blend_radius_m)
    |   movel([-0.100917, -1.454564, -2.519654, -0.738172, 1.570796, 1.469879],accel_mss,speed_ms,0,blend_radius_m)
    |   movel([-0.101020, -1.451573, -2.522084, -0.738731, 1.570796, 1.469776],accel_mss,speed_ms,0,blend_radius_m)
    |   movel([-0.100913, -1.448486, -2.524579, -0.739323, 1.570796, 1.469883],accel_mss,speed_ms,0,blend_radius_m)
    |   movel([-0.100604, -1.445317, -2.527125, -0.739946, 1.570796, 1.470192],accel_mss,speed_ms,0,blend_radius_m)
    |   movel([-0.100098, -1.442082, -2.529709, -0.740598, 1.570796, 1.470699],accel_mss,speed_ms,0,blend_radius_m)
    |   movel([-0.099400, -1.438790, -2.532321, -0.741278, 1.570796, 1.471396],accel_mss,speed_ms,0,blend_radius_m)
    |   movel([-0.098520, -1.435458, -2.534948, -0.741983, 1.570796, 1.472277],accel_mss,speed_ms,0,blend_radius_m)
    |   movel([-0.097464, -1.432102, -2.537577, -0.742710, 1.570796, 1.473332],accel_mss,speed_ms,0,blend_radius_m)
    |   movel([-0.096240, -1.428735, -2.540197, -0.743456, 1.570796, 1.474556],accel_mss,speed_ms,0,blend_radius_m)
    |   movel([-0.094858, -1.425377, -2.542794, -0.744218, 1.570796, 1.475938],accel_mss,speed_ms,0,blend_radius_m)
    |   movel([-0.093321, -1.422040, -2.545357, -0.744992, 1.570796, 1.477475],accel_mss,speed_ms,0,blend_radius_m)
    |   movel([-0.091642, -1.418741, -2.547874, -0.745773, 1.570796, 1.479154],accel_mss,speed_ms,0,blend_radius_m)
    |   movel([-0.088194, -1.412581, -2.552532, -0.747276, 1.570796, 1.482602],accel_mss,speed_ms,0,blend_radius_m)
    |   movel([-0.086308, -1.409493, -2.554845, -0.748051, 1.570796, 1.484489],accel_mss,speed_ms,0,blend_radius_m)
    |   movel([-0.084288, -1.406418, -2.557135, -0.748837, 1.570796, 1.486508],accel_mss,speed_ms,0,blend_radius_m)
    |   movel([-0.082113, -1.403371, -2.559390, -0.749629, 1.570796, 1.488683],accel_mss,speed_ms,0,blend_radius_m)
    |   movel([-0.079766, -1.400370, -2.561597, -0.750422, 1.570796, 1.491030],accel_mss,speed_ms,0,blend_radius_m)
    |   movel([-0.077228, -1.397430, -2.563747, -0.751213, 1.570796, 1.493568],accel_mss,speed_ms,0,blend_radius_m)
    |   movel([-0.074479, -1.394567, -2.565828, -0.751994, 1.570796, 1.496318],accel_mss,speed_ms,0,blend_radius_m)
    |   movel([-0.071202, -1.391495, -2.568047, -0.752847, 1.570796, 1.499594],accel_mss,speed_ms,0,blend_radius_m)
    |   movel([-0.067735, -1.388536, -2.570172, -0.753681, 1.570796, 1.503061],accel_mss,speed_ms,0,blend_radius_m)
    |   movel([-0.064098, -1.385698, -2.572199, -0.754493, 1.570796, 1.506698],accel_mss,speed_ms,0,blend_radius_m)
    |   movel([-0.060310, -1.382989, -2.574122, -0.755278, 1.570796, 1.510487],accel_mss,speed_ms,0,blend_radius_m)
    |   movel([-0.056391, -1.380420, -2.575936, -0.756033, 1.570796, 1.514405],accel_mss,speed_ms,0,blend_radius_m)
    |   movel([-0.052365, -1.377999, -2.577636, -0.756753, 1.570796, 1.518431],accel_mss,speed_ms,0,blend_radius_m)
    |   movel([-0.048248, -1.375735, -2.579219, -0.757435, 1.570796, 1.522548],accel_mss,speed_ms,0,blend_radius_m)
    |   movel([-0.044065, -1.373638, -2.580679, -0.758072, 1.570796, 1.526731],accel_mss,speed_ms,0,blend_radius_m)
    |   movel([-0.039838, -1.371718, -2.582010, -0.758661, 1.570796, 1.530959],accel_mss,speed_ms,0,blend_radius_m)
    |   movel([-0.035590, -1.369980, -2.583210, -0.759199, 1.570796, 1.535206],accel_mss,speed_ms,0,blend_radius_m)
    |   movel([-0.031342, -1.368436, -2.584273, -0.759681, 1.570796, 1.539455],accel_mss,speed_ms,0,blend_radius_m)
    |   movel([-0.027115, -1.367091, -2.585195, -0.760103, 1.570796, 1.543681],accel_mss,speed_ms,0,blend_radius_m)
    |   movel([-0.022938, -1.365954, -2.585973, -0.760462, 1.570796, 1.547859],accel_mss,speed_ms,0,blend_radius_m)
    |   movel([-0.018827, -1.365032, -2.586603, -0.760754, 1.570796, 1.551969],accel_mss,speed_ms,0,blend_radius_m)
    |   movel([-0.014807, -1.364330, -2.587081, -0.760977, 1.570796, 1.555989],accel_mss,speed_ms,0,blend_radius_m)
    |   movel([-0.010899, -1.363858, -2.587403, -0.761128, 1.570796, 1.559897],accel_mss,speed_ms,0,blend_radius_m)
    |   movel([-0.006829, -1.363541, -2.587618, -0.761229, 1.570796, 1.563967],accel_mss,speed_ms,0,blend_radius_m)
    |   movel([-0.002820, -1.363384, -2.587726, -0.761280, 1.570796, 1.567976],accel_mss,speed_ms,0,blend_radius_m)
    |   movel([0.001098, -1.363425, -2.587697, -0.761266, 1.570796, 1.571894],accel_mss,speed_ms,0,blend_radius_m)
    |   movel([0.004894, -1.363713, -2.587502, -0.761175, 1.570796, 1.575691],accel_mss,speed_ms,0,blend_radius_m)
    |   movel([0.009149, -1.364394, -2.587038, -0.760957, 1.570796, 1.579946],accel_mss,speed_ms,0,blend_radius_m)
    |   movel([0.013233, -1.365436, -2.586327, -0.760626, 1.570796, 1.584029],accel_mss,speed_ms,0,blend_radius_m)
    |   movel([0.017106, -1.366821, -2.585380, -0.760188, 1.570796, 1.587902],accel_mss,speed_ms,0,blend_radius_m)
    |   movel([0.020731, -1.368531, -2.584207, -0.759651, 1.570796, 1.591527],accel_mss,speed_ms,0,blend_radius_m)
    |   movel([0.024074, -1.370546, -2.582819, -0.759024, 1.570796, 1.594870],accel_mss,speed_ms,0,blend_radius_m)
    |   movel([0.027099, -1.372846, -2.581228, -0.758315, 1.570796, 1.597895],accel_mss,speed_ms,0,blend_radius_m)
    |   movel([0.029775, -1.375406, -2.579449, -0.757534, 1.570796, 1.600572],accel_mss,speed_ms,0,blend_radius_m)
    |   movel([0.032074, -1.378207, -2.577491, -0.756691, 1.570796, 1.602870],accel_mss,speed_ms,0,blend_radius_m)
    |   movel([0.036161, -1.384036, -2.573380, -0.754973, 1.570796, 1.606957],accel_mss,speed_ms,0,blend_radius_m)
    |   movel([0.038008, -1.387050, -2.571235, -0.754104, 1.570796, 1.608804],accel_mss,speed_ms,0,blend_radius_m)
    |   movel([0.039646, -1.390258, -2.568937, -0.753194, 1.570796, 1.610442],accel_mss,speed_ms,0,blend_radius_m)
    |   movel([0.042293, -1.395720, -2.564991, -0.751678, 1.570796, 1.613089],accel_mss,speed_ms,0,blend_radius_m)
    |   movel([0.043799, -1.398370, -2.563061, -0.750959, 1.570796, 1.614595],accel_mss,speed_ms,0,blend_radius_m)
    |   movel([0.045476, -1.400889, -2.561216, -0.750284, 1.570796, 1.616272],accel_mss,speed_ms,0,blend_radius_m)
    |   movel([0.047368, -1.403223, -2.559499, -0.749667, 1.570796, 1.618164],accel_mss,speed_ms,0,blend_radius_m)
    |   movel([0.049508, -1.405317, -2.557951, -0.749121, 1.570796, 1.620304],accel_mss,speed_ms,0,blend_radius_m)
    |   movel([0.051940, -1.407117, -2.556616, -0.748657, 1.570796, 1.622736],accel_mss,speed_ms,0,blend_radius_m)
    |   movel([0.054700, -1.408569, -2.555535, -0.748286, 1.570796, 1.625496],accel_mss,speed_ms,0,blend_radius_m)
    |   movel([0.055929, -1.409007, -2.555208, -0.748174, 1.570796, 1.626726],accel_mss,speed_ms,0,blend_radius_m)
    |   movel([0.057287, -1.409249, -2.555027, -0.748113, 1.570796, 1.628084],accel_mss,speed_ms,0,blend_radius_m)
    |   movel([0.058007, -1.409257, -2.555021, -0.748111, 1.570796, 1.628803],accel_mss,speed_ms,0,blend_radius_m)
    |   movel([0.058747, -1.409170, -2.555086, -0.748133, 1.570796, 1.629544],accel_mss,speed_ms,0,blend_radius_m)
    |   movel([0.059507, -1.408974, -2.555233, -0.748183, 1.570796, 1.630304],accel_mss,speed_ms,0,blend_radius_m)
    |   movel([0.060279, -1.408650, -2.555474, -0.748265, 1.570796, 1.631075],accel_mss,speed_ms,0,blend_radius_m)
    |   movel([0.061049, -1.408194, -2.555814, -0.748381, 1.570796, 1.631845],accel_mss,speed_ms,0,blend_radius_m)
    |   movel([0.061762, -1.407642, -2.556225, -0.748522, 1.570796, 1.632558],accel_mss,speed_ms,0,blend_radius_m)
    |   movel([0.063014, -1.406358, -2.557179, -0.748852, 1.570796, 1.633811],accel_mss,speed_ms,0,blend_radius_m)
    |   movel([0.063753, -1.405394, -2.557894, -0.749101, 1.570796, 1.634550],accel_mss,speed_ms,0,blend_radius_m)
    |   movel([0.064381, -1.404409, -2.558623, -0.749357, 1.570796, 1.635177],accel_mss,speed_ms,0,blend_radius_m)
    |   movel([0.065330, -1.402399, -2.560106, -0.749884, 1.570796, 1.636126],accel_mss,speed_ms,0,blend_radius_m)
    |   movel([0.065915, -1.400362, -2.561603, -0.750424, 1.570796, 1.636712],accel_mss,speed_ms,0,blend_radius_m)
    |   movel([0.066194, -1.398329, -2.563090, -0.750970, 1.570796, 1.636991],accel_mss,speed_ms,0,blend_radius_m)
    |   movel([0.066220, -1.396340, -2.564540, -0.751509, 1.570796, 1.637016],accel_mss,speed_ms,0,blend_radius_m)
    |   movel([0.066047, -1.394428, -2.565928, -0.752033, 1.570796, 1.636844],accel_mss,speed_ms,0,blend_radius_m)
    |   movel([0.065732, -1.392629, -2.567230, -0.752531, 1.570796, 1.636528],accel_mss,speed_ms,0,blend_radius_m)
    |   movel([0.064746, -1.389183, -2.569709, -0.753497, 1.570796, 1.635542],accel_mss,speed_ms,0,blend_radius_m)
    |   movel([0.064002, -1.387475, -2.570931, -0.753983, 1.570796, 1.634799],accel_mss,speed_ms,0,blend_radius_m)
    |   movel([0.063104, -1.385861, -2.572082, -0.754446, 1.570796, 1.633900],accel_mss,speed_ms,0,blend_radius_m)
    |   movel([0.062052, -1.384355, -2.573153, -0.754881, 1.570796, 1.632848],accel_mss,speed_ms,0,blend_radius_m)
    |   movel([0.060847, -1.382961, -2.574142, -0.755287, 1.570796, 1.631643],accel_mss,speed_ms,0,blend_radius_m)
    |   movel([0.059493, -1.381691, -2.575039, -0.755658, 1.570796, 1.630289],accel_mss,speed_ms,0,blend_radius_m)
    |   movel([0.057997, -1.380552, -2.575842, -0.755994, 1.570796, 1.628794],accel_mss,speed_ms,0,blend_radius_m)
    |   movel([0.056359, -1.379553, -2.576545, -0.756290, 1.570796, 1.627155],accel_mss,speed_ms,0,blend_radius_m)
    |   speed_ms = 0.005
    |   movel([0.056359, -1.370765, -2.572549, -0.769076, 1.570796, 1.627155],accel_mss,speed_ms,0,blend_radius_m)
    |   speed_ms = 0.040
    |   movel([0.056256, -1.386026, -2.561797, -0.764566, 1.570796, 1.627052],accel_mss,speed_ms,0,blend_radius_m)
    |   speed_ms = 0.005
    |   movel([0.056256, -1.394705, -2.565727, -0.751956, 1.570796, 1.627052],accel_mss,speed_ms,0,blend_radius_m)
    |   speed_ms = 0.025
    |   movel([0.054176, -1.393655, -2.566488, -0.752246, 1.570796, 1.624973],accel_mss,speed_ms,0,blend_radius_m)
    |   movel([0.051871, -1.392874, -2.567053, -0.752462, 1.570796, 1.622668],accel_mss,speed_ms,0,blend_radius_m)
    |   movel([0.050615, -1.392653, -2.567212, -0.752524, 1.570796, 1.621411],accel_mss,speed_ms,0,blend_radius_m)
    |   movel([0.049282, -1.392584, -2.567262, -0.752543, 1.570796, 1.620078],accel_mss,speed_ms,0,blend_radius_m)
    |   movel([0.047868, -1.392691, -2.567184, -0.752513, 1.570796, 1.618664],accel_mss,speed_ms,0,blend_radius_m)
    |   movel([0.046364, -1.393002, -2.566960, -0.752427, 1.570796, 1.617160],accel_mss,speed_ms,0,blend_radius_m)
    |   speed_ms = 0.005
    |   movel([0.046364, -1.384310, -2.563022, -0.765057, 1.570796, 1.617160],accel_mss,speed_ms,0,blend_radius_m)
    |   speed_ms = 0.040
    |   movel([0.050800, -1.379714, -2.566284, -0.766391, 1.570796, 1.621596],accel_mss,speed_ms,0,blend_radius_m)
    |   speed_ms = 0.005
    |   movel([0.050800, -1.388439, -2.570242, -0.753708, 1.570796, 1.621596],accel_mss,speed_ms,0,blend_radius_m)
    |   speed_ms = 0.025
    |   movel([0.050701, -1.386443, -2.571668, -0.754278, 1.570796, 1.621498],accel_mss,speed_ms,0,blend_radius_m)
    |   movel([0.050175, -1.384681, -2.572921, -0.754786, 1.570796, 1.620971],accel_mss,speed_ms,0,blend_radius_m)
    |   movel([0.049255, -1.383178, -2.573988, -0.755223, 1.570796, 1.620052],accel_mss,speed_ms,0,blend_radius_m)
    |   movel([0.047974, -1.381967, -2.574845, -0.755578, 1.570796, 1.618770],accel_mss,speed_ms,0,blend_radius_m)
    |   movel([0.046366, -1.381074, -2.575475, -0.755840, 1.570796, 1.617163],accel_mss,speed_ms,0,blend_radius_m)
    |   movel([0.044470, -1.380530, -2.575858, -0.756001, 1.570796, 1.615267],accel_mss,speed_ms,0,blend_radius_m)
    |   movel([0.042323, -1.380360, -2.575978, -0.756051, 1.570796, 1.613120],accel_mss,speed_ms,0,blend_radius_m)
    |   movel([0.041166, -1.380425, -2.575932, -0.756032, 1.570796, 1.611962],accel_mss,speed_ms,0,blend_radius_m)
    |   movel([0.039961, -1.380591, -2.575815, -0.755983, 1.570796, 1.610757],accel_mss,speed_ms,0,blend_radius_m)
    |   speed_ms = 0.005
    |   movel([0.039961, -1.371810, -2.571823, -0.768756, 1.570796, 1.610757],accel_mss,speed_ms,0,blend_radius_m)
    |   speed_ms = 0.040
    |   movel([0.045655, -1.367633, -2.574714, -0.770042, 1.570796, 1.616452],accel_mss,speed_ms,0,blend_radius_m)
    |   speed_ms = 0.005
    |   movel([0.045655, -1.376444, -2.578724, -0.757221, 1.570796, 1.616452],accel_mss,speed_ms,0,blend_radius_m)
    |   speed_ms = 0.025
    |   movel([0.045426, -1.375518, -2.579371, -0.757501, 1.570796, 1.616223],accel_mss,speed_ms,0,blend_radius_m)
    |   movel([0.045059, -1.374646, -2.579978, -0.757765, 1.570796, 1.615855],accel_mss,speed_ms,0,blend_radius_m)
    |   movel([0.043947, -1.373084, -2.581063, -0.758242, 1.570796, 1.614743],accel_mss,speed_ms,0,blend_radius_m)
    |   movel([0.042397, -1.371794, -2.581957, -0.758638, 1.570796, 1.613193],accel_mss,speed_ms,0,blend_radius_m)
    |   movel([0.040492, -1.370817, -2.582633, -0.758940, 1.570796, 1.611289],accel_mss,speed_ms,0,blend_radius_m)
    |   movel([0.038312, -1.370180, -2.583072, -0.759137, 1.570796, 1.609108],accel_mss,speed_ms,0,blend_radius_m)
    |   movel([0.035947, -1.369917, -2.583253, -0.759219, 1.570796, 1.606743],accel_mss,speed_ms,0,blend_radius_m)
    |   movel([0.034719, -1.369938, -2.583239, -0.759212, 1.570796, 1.605515],accel_mss,speed_ms,0,blend_radius_m)
    |   movel([0.032231, -1.370296, -2.582992, -0.759101, 1.570796, 1.603027],accel_mss,speed_ms,0,blend_radius_m)
    |   movel([0.030992, -1.370640, -2.582755, -0.758995, 1.570796, 1.601788],accel_mss,speed_ms,0,blend_radius_m)
    |   speed_ms = 0.005
    |   movel([0.030992, -1.361788, -2.578719, -0.771882, 1.570796, 1.601788],accel_mss,speed_ms,0,blend_radius_m)
    |   speed_ms = 0.040
    |   movel([0.039126, -1.356851, -2.582064, -0.773474, 1.570796, 1.609923],accel_mss,speed_ms,0,blend_radius_m)
    |   speed_ms = 0.005
    |   movel([0.039126, -1.365737, -2.586122, -0.760531, 1.570796, 1.609923],accel_mss,speed_ms,0,blend_radius_m)
    |   speed_ms = 0.025
    |   movel([0.037538, -1.364150, -2.587204, -0.761035, 1.570796, 1.608334],accel_mss,speed_ms,0,blend_radius_m)
    |   movel([0.035621, -1.362863, -2.588079, -0.761446, 1.570796, 1.606418],accel_mss,speed_ms,0,blend_radius_m)
    |   movel([0.033416, -1.361920, -2.588719, -0.761750, 1.570796, 1.604213],accel_mss,speed_ms,0,blend_radius_m)
    |   movel([0.030951, -1.361352, -2.589104, -0.761933, 1.570796, 1.601747],accel_mss,speed_ms,0,blend_radius_m)
    |   movel([0.028264, -1.361199, -2.589207, -0.761982, 1.570796, 1.599060],accel_mss,speed_ms,0,blend_radius_m)
    |   movel([0.026848, -1.361288, -2.589147, -0.761954, 1.570796, 1.597645],accel_mss,speed_ms,0,blend_radius_m)
    |   movel([0.025393, -1.361494, -2.589008, -0.761887, 1.570796, 1.596189],accel_mss,speed_ms,0,blend_radius_m)
    |   movel([0.023898, -1.361820, -2.588787, -0.761782, 1.570796, 1.594695],accel_mss,speed_ms,0,blend_radius_m)
    |   movel([0.022370, -1.362271, -2.588481, -0.761637, 1.570796, 1.593166],accel_mss,speed_ms,0,blend_radius_m)
    |   movel([0.020816, -1.362849, -2.588089, -0.761451, 1.570796, 1.591612],accel_mss,speed_ms,0,blend_radius_m)
    |   movel([0.019239, -1.363559, -2.587606, -0.761224, 1.570796, 1.590036],accel_mss,speed_ms,0,blend_radius_m)
    |   speed_ms = 0.005
    |   movel([0.019239, -1.354658, -2.583539, -0.774192, 1.570796, 1.590036],accel_mss,speed_ms,0,blend_radius_m)
    |   speed_ms = 0.040
    |   movel([0.027863, -1.348222, -2.587830, -0.776338, 1.570796, 1.598660],accel_mss,speed_ms,0,blend_radius_m)
    |   speed_ms = 0.005
    |   movel([0.027863, -1.357166, -2.591926, -0.763297, 1.570796, 1.598660],accel_mss,speed_ms,0,blend_radius_m)
    |   speed_ms = 0.025
    |   movel([0.027318, -1.355873, -2.592792, -0.763723, 1.570796, 1.598114],accel_mss,speed_ms,0,blend_radius_m)
    |   movel([0.026528, -1.354745, -2.593546, -0.764097, 1.570796, 1.597324],accel_mss,speed_ms,0,blend_radius_m)
    |   movel([0.025508, -1.353804, -2.594174, -0.764410, 1.570796, 1.596304],accel_mss,speed_ms,0,blend_radius_m)
    |   movel([0.024278, -1.353073, -2.594661, -0.764655, 1.570796, 1.595074],accel_mss,speed_ms,0,blend_radius_m)
    |   movel([0.022555, -1.352476, -2.595058, -0.764855, 1.570796, 1.593351],accel_mss,speed_ms,0,blend_radius_m)
    |   movel([0.020651, -1.352134, -2.595285, -0.764969, 1.570796, 1.591447],accel_mss,speed_ms,0,blend_radius_m)
    |   movel([0.018265, -1.351979, -2.595389, -0.765022, 1.570796, 1.589062],accel_mss,speed_ms,0,blend_radius_m)
    |   movel([0.015752, -1.352104, -2.595306, -0.764980, 1.570796, 1.586548],accel_mss,speed_ms,0,blend_radius_m)
    |   movel([0.013143, -1.352538, -2.595017, -0.764834, 1.570796, 1.583939],accel_mss,speed_ms,0,blend_radius_m)
    |   movel([0.010469, -1.353317, -2.594499, -0.764573, 1.570796, 1.581266],accel_mss,speed_ms,0,blend_radius_m)
    |   movel([0.007776, -1.354471, -2.593729, -0.764188, 1.570796, 1.578573],accel_mss,speed_ms,0,blend_radius_m)
    |   movel([0.006451, -1.355185, -2.593253, -0.763951, 1.570796, 1.577247],accel_mss,speed_ms,0,blend_radius_m)
    |   movel([0.003913, -1.356864, -2.592129, -0.763397, 1.570796, 1.574709],accel_mss,speed_ms,0,blend_radius_m)
    |   movel([0.002724, -1.357817, -2.591488, -0.763083, 1.570796, 1.573520],accel_mss,speed_ms,0,blend_radius_m)
    |   movel([0.001609, -1.358842, -2.590799, -0.762748, 1.570796, 1.572406],accel_mss,speed_ms,0,blend_radius_m)
    |   movel([0.000580, -1.359933, -2.590063, -0.762392, 1.570796, 1.571376],accel_mss,speed_ms,0,blend_radius_m)
    |   speed_ms = 0.005
    |   movel([0.000580, -1.351007, -2.585980, -0.775402, 1.570796, 1.571376],accel_mss,speed_ms,0,blend_radius_m)
    |   speed_ms = 0.040
    |   movel([0.009787, -1.340894, -2.592645, -0.778850, 1.570796, 1.580584],accel_mss,speed_ms,0,blend_radius_m)
    |   speed_ms = 0.005
    |   movel([0.009787, -1.349888, -2.596774, -0.765727, 1.570796, 1.580584],accel_mss,speed_ms,0,blend_radius_m)
    |   speed_ms = 0.025
    |   movel([0.006644, -1.349839, -2.596806, -0.765744, 1.570796, 1.577440],accel_mss,speed_ms,0,blend_radius_m)
    |   movel([0.003301, -1.350135, -2.596610, -0.765644, 1.570796, 1.574097],accel_mss,speed_ms,0,blend_radius_m)
    |   movel([-0.000160, -1.350811, -2.596163, -0.765415, 1.570796, 1.570637],accel_mss,speed_ms,0,blend_radius_m)
    |   movel([-0.001908, -1.351297, -2.595841, -0.765251, 1.570796, 1.568888],accel_mss,speed_ms,0,blend_radius_m)
    |   movel([-0.003655, -1.351890, -2.595448, -0.765052, 1.570796, 1.567141],accel_mss,speed_ms,0,blend_radius_m)
    |   movel([-0.005388, -1.352589, -2.594983, -0.764817, 1.570796, 1.565409],accel_mss,speed_ms,0,blend_radius_m)
    |   movel([-0.007094, -1.353398, -2.594445, -0.764546, 1.570796, 1.563702],accel_mss,speed_ms,0,blend_radius_m)
    |   movel([-0.008766, -1.354321, -2.593829, -0.764238, 1.570796, 1.562031],accel_mss,speed_ms,0,blend_radius_m)
    |   movel([-0.010392, -1.355362, -2.593134, -0.763893, 1.570796, 1.560405],accel_mss,speed_ms,0,blend_radius_m)
    |   movel([-0.011963, -1.356521, -2.592359, -0.763510, 1.570796, 1.558833],accel_mss,speed_ms,0,blend_radius_m)
    |   movel([-0.013464, -1.357801, -2.591499, -0.763088, 1.570796, 1.557332],accel_mss,speed_ms,0,blend_radius_m)
    |   movel([-0.014889, -1.359205, -2.590555, -0.762630, 1.570796, 1.555907],accel_mss,speed_ms,0,blend_radius_m)
    |   movel([-0.016224, -1.360736, -2.589521, -0.762132, 1.570796, 1.554572],accel_mss,speed_ms,0,blend_radius_m)
    |   speed_ms = 0.005
    |   movel([-0.016224, -1.351815, -2.585441, -0.775133, 1.570796, 1.554572],accel_mss,speed_ms,0,blend_radius_m)
    |   speed_ms = 0.040
    |   movel([-0.009624, -1.340342, -2.593005, -0.779042, 1.570796, 1.561172],accel_mss,speed_ms,0,blend_radius_m)
    |   speed_ms = 0.005
    |   movel([-0.009624, -1.349340, -2.597136, -0.765913, 1.570796, 1.561172],accel_mss,speed_ms,0,blend_radius_m)
    |   speed_ms = 0.025
    |   movel([-0.011251, -1.349433, -2.597074, -0.765882, 1.570796, 1.559545],accel_mss,speed_ms,0,blend_radius_m)
    |   movel([-0.012933, -1.349679, -2.596912, -0.765798, 1.570796, 1.557864],accel_mss,speed_ms,0,blend_radius_m)
    |   movel([-0.014648, -1.350076, -2.596650, -0.765664, 1.570796, 1.556148],accel_mss,speed_ms,0,blend_radius_m)
    |   movel([-0.016385, -1.350614, -2.596294, -0.765482, 1.570796, 1.554412],accel_mss,speed_ms,0,blend_radius_m)
    |   movel([-0.018128, -1.351290, -2.595846, -0.765254, 1.570796, 1.552669],accel_mss,speed_ms,0,blend_radius_m)
    |   movel([-0.019858, -1.352097, -2.595310, -0.764982, 1.570796, 1.550938],accel_mss,speed_ms,0,blend_radius_m)
    |   movel([-0.021560, -1.353028, -2.594691, -0.764670, 1.570796, 1.549236],accel_mss,speed_ms,0,blend_radius_m)
    |   movel([-0.023221, -1.354078, -2.593992, -0.764319, 1.570796, 1.547575],accel_mss,speed_ms,0,blend_radius_m)
    |   movel([-0.024821, -1.355239, -2.593217, -0.763933, 1.570796, 1.545975],accel_mss,speed_ms,0,blend_radius_m)
    |   movel([-0.026346, -1.356495, -2.592376, -0.763518, 1.570796, 1.544450],accel_mss,speed_ms,0,blend_radius_m)
    |   movel([-0.027783, -1.357833, -2.591478, -0.763078, 1.570796, 1.543013],accel_mss,speed_ms,0,blend_radius_m)
    |   movel([-0.029122, -1.359241, -2.590530, -0.762618, 1.570796, 1.541674],accel_mss,speed_ms,0,blend_radius_m)
    |   movel([-0.030353, -1.360704, -2.589543, -0.762143, 1.570796, 1.540443],accel_mss,speed_ms,0,blend_radius_m)
    |   movel([-0.031466, -1.362211, -2.588522, -0.761656, 1.570796, 1.539331],accel_mss,speed_ms,0,blend_radius_m)
    |   movel([-0.032443, -1.363746, -2.587479, -0.761164, 1.570796, 1.538354],accel_mss,speed_ms,0,blend_radius_m)
    |   movel([-0.033280, -1.365298, -2.586422, -0.760670, 1.570796, 1.537516],accel_mss,speed_ms,0,blend_radius_m)
    |   speed_ms = 0.005
    |   movel([-0.033280, -1.356409, -2.582362, -0.773618, 1.570796, 1.537516],accel_mss,speed_ms,0,blend_radius_m)
    |   speed_ms = 0.040
    |   movel([-0.029508, -1.345457, -2.589655, -0.777277, 1.570796, 1.541288],accel_mss,speed_ms,0,blend_radius_m)
    |   speed_ms = 0.005
    |   movel([-0.029508, -1.354421, -2.593763, -0.764205, 1.570796, 1.541288],accel_mss,speed_ms,0,blend_radius_m)
    |   speed_ms = 0.025
    |   movel([-0.031119, -1.354616, -2.593633, -0.764140, 1.570796, 1.539678],accel_mss,speed_ms,0,blend_radius_m)
    |   movel([-0.032775, -1.355067, -2.593332, -0.763991, 1.570796, 1.538021],accel_mss,speed_ms,0,blend_radius_m)
    |   movel([-0.034448, -1.355742, -2.592880, -0.763767, 1.570796, 1.536348],accel_mss,speed_ms,0,blend_radius_m)
    |   movel([-0.036120, -1.356609, -2.592299, -0.763480, 1.570796, 1.534677],accel_mss,speed_ms,0,blend_radius_m)
    |   movel([-0.037765, -1.357638, -2.591609, -0.763142, 1.570796, 1.533031],accel_mss,speed_ms,0,blend_radius_m)
    |   movel([-0.039359, -1.358795, -2.590831, -0.762763, 1.570796, 1.531437],accel_mss,speed_ms,0,blend_radius_m)
    |   movel([-0.040885, -1.360047, -2.589986, -0.762356, 1.570796, 1.529911],accel_mss,speed_ms,0,blend_radius_m)
    |   movel([-0.042314, -1.361365, -2.589095, -0.761929, 1.570796, 1.528483],accel_mss,speed_ms,0,blend_radius_m)
    |   movel([-0.043694, -1.362780, -2.588136, -0.761473, 1.570796, 1.527102],accel_mss,speed_ms,0,blend_radius_m)
    |   movel([-0.044980, -1.364256, -2.587132, -0.761001, 1.570796, 1.525816],accel_mss,speed_ms,0,blend_radius_m)
    |   movel([-0.046152, -1.365777, -2.586094, -0.760518, 1.570796, 1.524645],accel_mss,speed_ms,0,blend_radius_m)
    |   movel([-0.047176, -1.367326, -2.585034, -0.760029, 1.570796, 1.523620],accel_mss,speed_ms,0,blend_radius_m)
    |   movel([-0.048032, -1.368882, -2.583966, -0.759541, 1.570796, 1.522765],accel_mss,speed_ms,0,blend_radius_m)
    |   movel([-0.048694, -1.370427, -2.582901, -0.759060, 1.570796, 1.522103],accel_mss,speed_ms,0,blend_radius_m)
    |   movel([-0.049130, -1.371946, -2.581852, -0.758591, 1.570796, 1.521666],accel_mss,speed_ms,0,blend_radius_m)
    |   movel([-0.049322, -1.373418, -2.580832, -0.758139, 1.570796, 1.521474],accel_mss,speed_ms,0,blend_radius_m)
    |   speed_ms = 0.005
    |   movel([-0.049322, -1.364586, -2.576808, -0.770995, 1.570796, 1.521474],accel_mss,speed_ms,0,blend_radius_m)
    |   speed_ms = 0.040
    |   movel([-0.049808, -1.355807, -2.582767, -0.773815, 1.570796, 1.520988],accel_mss,speed_ms,0,blend_radius_m)
    |   speed_ms = 0.005
    |   movel([-0.049808, -1.364700, -2.586829, -0.760859, 1.570796, 1.520988],accel_mss,speed_ms,0,blend_radius_m)
    |   speed_ms = 0.025
    |   movel([-0.052106, -1.366060, -2.585901, -0.760428, 1.570796, 1.518691],accel_mss,speed_ms,0,blend_radius_m)
    |   movel([-0.054439, -1.367711, -2.584770, -0.759908, 1.570796, 1.516358],accel_mss,speed_ms,0,blend_radius_m)
    |   movel([-0.056681, -1.369587, -2.583480, -0.759321, 1.570796, 1.514116],accel_mss,speed_ms,0,blend_radius_m)
    |   movel([-0.058703, -1.371619, -2.582078, -0.758692, 1.570796, 1.512093],accel_mss,speed_ms,0,blend_radius_m)
    |   movel([-0.060386, -1.373741, -2.580607, -0.758041, 1.570796, 1.510411],accel_mss,speed_ms,0,blend_radius_m)
    |   movel([-0.061062, -1.374817, -2.579859, -0.757713, 1.570796, 1.509735],accel_mss,speed_ms,0,blend_radius_m)
    |   movel([-0.061605, -1.375890, -2.579111, -0.757388, 1.570796, 1.509191],accel_mss,speed_ms,0,blend_radius_m)
    |   movel([-0.062005, -1.376955, -2.578367, -0.757067, 1.570796, 1.508792],accel_mss,speed_ms,0,blend_radius_m)
    |   movel([-0.062245, -1.378004, -2.577633, -0.756752, 1.570796, 1.508551],accel_mss,speed_ms,0,blend_radius_m)
    |   movel([-0.062307, -1.379024, -2.576917, -0.756447, 1.570796, 1.508490],accel_mss,speed_ms,0,blend_radius_m)
    |   movel([-0.062180, -1.380016, -2.576220, -0.756153, 1.570796, 1.508616],accel_mss,speed_ms,0,blend_radius_m)
    |   speed_ms = 0.005
    |   movel([-0.062180, -1.371230, -2.572225, -0.768933, 1.570796, 1.508616],accel_mss,speed_ms,0,blend_radius_m)
    |   speed_ms = 0.040
    |   movel([-0.066185, -1.368693, -2.573983, -0.769713, 1.570796, 1.504611],accel_mss,speed_ms,0,blend_radius_m)
    |   speed_ms = 0.005
    |   movel([-0.066185, -1.377496, -2.577989, -0.756904, 1.570796, 1.504611],accel_mss,speed_ms,0,blend_radius_m)
    |   speed_ms = 0.025
    |   movel([-0.068894, -1.380459, -2.575908, -0.756022, 1.570796, 1.501902],accel_mss,speed_ms,0,blend_radius_m)
    |   movel([-0.070132, -1.382012, -2.574813, -0.755564, 1.570796, 1.500664],accel_mss,speed_ms,0,blend_radius_m)
    |   movel([-0.071233, -1.383588, -2.573697, -0.755104, 1.570796, 1.499563],accel_mss,speed_ms,0,blend_radius_m)
    |   movel([-0.072155, -1.385178, -2.572568, -0.754642, 1.570796, 1.498642],accel_mss,speed_ms,0,blend_radius_m)
    |   movel([-0.072857, -1.386769, -2.571435, -0.754185, 1.570796, 1.497939],accel_mss,speed_ms,0,blend_radius_m)
    |   movel([-0.073294, -1.388344, -2.570309, -0.753735, 1.570796, 1.497502],accel_mss,speed_ms,0,blend_radius_m)
    |   movel([-0.073429, -1.389895, -2.569198, -0.753296, 1.570796, 1.497368],accel_mss,speed_ms,0,blend_radius_m)
    |   speed_ms = 0.005
    |   # Splitting Linear movement in 2 (instruction 3386: MoveL 3110)
    |   movel([-0.073429, -1.368405, -2.559208, -0.784776, 1.570796, 1.497368],accel_mss,speed_ms,0,blend_radius_m)
    |   movel([-0.073429, -1.347892, -2.548856, -0.815641, 1.570796, 1.497368],accel_mss,speed_ms,0,blend_radius_m)
    |   speed_ms = 1.000
    |   movel([-0.073429, -1.347892, -2.548856, -0.815641, 1.570796, 1.497368],accel_mss,speed_ms,0,blend_radius_m)
    |   # Splitting Linear movement in 2 (instruction 3389: MoveL 3112)
    |   movel([-0.073429, -1.318924, -2.532681, -0.860784, 1.570796, 1.497368],accel_mss,speed_ms,0,blend_radius_m)
    |   movel([-0.073429, -1.292060, -2.515776, -0.904553, 1.570796, 1.497368],accel_mss,speed_ms,0,blend_radius_m)
    |   # End of main program
    | end
    | 
    | Machining2()
